// LS Electric XG5000 project: test_8.19
// PLC LSPLC

PROGRAM NewProgram (task: 스캔 프로그램)

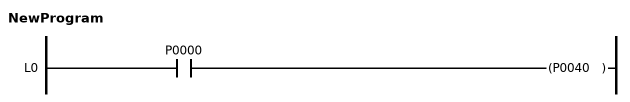
; L0
LOAD      P0000
OUT       P0040